TYPE EL3078_CHANNEL :
STRUCT
	Status AT %I* : WORD;
	Value AT %I* : REAL;
END_STRUCT
END_TYPE

(* stored: Version 1.1.0.1, ProductVersion 3.1.4026.18
   DUT EL3078_CHANNEL: Id {4361d0c9-c2d1-4cff-b4d0-bc2e9ae63f5c} *)
